Staubli VAL3: onF1Event.pgx

program onF1Event(bool& x_bSave[])
  local string l_sParameter
  local string l_sItem
  local num l_nKey
  local num l_nIndex
  local string l_sPage
  local string l_sEvent
  local num i
begin
  // look if the bButton is enable
  if bButton[0]
    //
    // TOOL / FRAME SELECTION
    //
    call use:setSizeList(0,9,10,2)
    call use:listcreate("")
    // TOOL
    call language:message(l_sItem,124)
    call use:listadd(l_sItem)
    l_sItem="FRAME"
    call use:listadd(l_sItem)
    call use:listupdate(0)
    // get the key
    do
      l_nKey=get()
      call use:listevent(l_nKey,l_nIndex,l_sEvent)
    until l_nKey==270 or l_nKey==255
    // check the Enter key pressure
    if l_nKey==270
      switch l_nIndex
        case 0
          // Select the tool
          l_sPage="Disk://kernel/page/tool"
          call loadPage(l_sPage,l_sItem)
        break
        case 1
          // Select the Frame
          l_sPage="Disk://kernel/page/frame"
          call loadPage(l_sPage,l_sItem)
        break
      endSwitch
    endIf
    logMsg("[KERNEL] INTERFACE:PAGE Advance")
    x_bSave=true
  endIf
end
